{attribute 'qualified_only'}
//{attribute 'strict'}
TYPE E_CX_HWType :
(
	//E_HW_UNKNOWN,
	CX1,
	CX2,
	CX5,
	CX8,
	CX9,
	CP,
	PC
);
END_TYPE

(* stored: Version 1.1.0.1
   DUT E_CX_HWType: Id {40d9759e-0b5a-4965-b4c4-96cd94ad58ed} *)
